FUNCTION_BLOCK Compressor (* Composite Function Block Type *)
  (* Standard: 61499-2 *)
  (* Version 0.0, 8/26/2024, SESA713705, Schneider Electric, template *)
  PACKAGE SE.Nereda;
  (* 00 - INITIALIZATION *)
  (* 06 - HMI INTERFACE *)
  (* 07- Input Hardware Interface *)
  FBS
    INIT : plcStart(Prio := 68, Delay := T#0ms);
    IThis : Compressor_HMI(QI := TRUE);
    Run : dISignal(Name := '$${PATH}DIn');
    Alarm : dISignal(Name := '$${PATH}DIn');
    Mode : dISignal(Name := '$${PATH}DIn');
    Frequency : aISignal(Name := '$${PATH}AIn');
    Power : aISignal(Name := '$${PATH}AIn');
    Capacity : aISignal(Name := '$${PATH}AIn');
  END_FBS
  EVENT_CONNECTIONS
    INIT.FIRST_INIT TO IThis.AD268C9638E5DBF1;
    INIT.REDO_INIT TO IThis.AD268C9638E5DBF1;
    Run.CNF TO IThis.2E55C76A903DF86E;
    Alarm.CNF TO IThis.2E55C76A903DF86E;
    Mode.CNF TO IThis.2E55C76A903DF86E;
    IThis.8C4D07A314DA5DB8 TO IThis.2E55C76A903DF86E;
    Frequency.CNF TO IThis.2E55C76A903DF86E;
    Power.CNF TO IThis.2E55C76A903DF86E;
    Capacity.CNF TO IThis.2E55C76A903DF86E;
    IThis.8C4D07A314DA5DB8 TO INIT.ACK_FIRST;
  END_CONNECTIONS
  DATA_CONNECTIONS
    Run.Out TO IThis.190C05C24FEBAA80;
    Alarm.Out TO IThis.2645D8C5BBB7C330;
    Mode.Out TO IThis.74773982CB014525;
    Frequency.Out TO IThis.3BDDF5275529359B;
    Power.Out TO IThis.EEF7C78472734FB1;
    Capacity.Out TO IThis.D5594589EE24C8C1;
  END_CONNECTIONS
END_FUNCTION_BLOCK
